PROGRAM Serial
VAR
    (*
    fbPfeifferSerialDriver : FB_PfeifferSerialDriver;
    fbPolling : TON;
    stPfeifferControl : lclsvacuumserialdriverlib.ST_PfeifferControl := (
        xEnableComm:= TRUE,
        iSerialAddress:= 0
        //xPumpingStation_010:= ,
        //xMotorPump_023:= ,
        //iGasMode_027:= ,
        //xIlk:= ,
        //xRunSW:= ,
        //xErrorAck_009:= ,
        //uiPowerPct_708:=
    );
    stRxBuffer : ComBuffer;
    stTxBuffer : ComBuffer;*)
END_VAR
VAR CONSTANT
    POLL_RATE : TIME := T#100MS;
    TIMEOUT : TIME := T#5S;
END_VAR

(*
fbPolling(IN := fbPfeifferSerialDriver.q_xDone, PT := POLL_RATE);

fbPfeifferSerialDriver(
    i_xExecute := fbPolling.Q,
    i_tTimeOut := TIMEOUT,
    i_stControl := stPfeifferControl,
    iq_stSerialRXBuffer := stRxBuffer,
    iq_stSerialTXBuffer := stTxBuffer);
*)

END_PROGRAM

(* stored: Version 1.1.0.1, ProductVersion 3.1.4022.17
   POU Serial: Id {893f175e-5a5c-4e2a-a383-b460a32427d2}, SpecialFunc None *)
